TYPE ST_CNCVariablesViewer_Data :
STRUCT
	strName : STRING;
	strValue  : STRING(127);
END_STRUCT
END_TYPE

(* stored: Version 1.1.0.1, ProductVersion 3.1.4019.0
   DUT ST_CNCVariablesViewer_Data: Id {2ec79d08-9304-4826-b236-00325e575ee4} *)
